// Mitsubishi GX Works2 project: CydeusPlatform   PLC: FX3U/FX3UC
// Cydeus Mitsu Platform

// global labels: GVL_Main
VAR_GLOBAL
  bAlarmTrigger AT M0 : BOOL;
  bManualMode AT M1 : BOOL;
  bAutoMode AT M2 : BOOL;
  bStepMode AT M3 : BOOL;
END_VAR

// global labels: GVL_Alarm
VAR_GLOBAL
  bMachineError AT M400 : BOOL;
  arrError AT M410 : ARRAY [0..9] OF BOOL;
  bResetError AT M401 : BOOL;
END_VAR
VAR_GLOBAL CONSTANT
  uiNumErrMinus1 : INT := 9;
END_VAR

// global labels: GVL_Output
VAR_GLOBAL
  bPunchingOutput AT Y006 : BOOL;
  bPowerMotor AT Y007 : BOOL;
END_VAR

// global labels: GVL_HMI
VAR_GLOBAL
  btnPunchingOutput : BOOL;
  btnPowerMotor : BOOL;
  btnManualMode : BOOL;
  btnInitialize : BOOL;
  btnAutoMode : BOOL;
  btnAbort : BOOL;
  btnStepMode : BOOL;
  btnBack : BOOL;
  btnTest : BOOL;
  btnTestManualOn : BOOL;
  btnSetup : BOOL;
END_VAR

// task Task_01 (event TRUE, interval 0, priority 31): MAIN

PROGRAM MAIN
VAR
  fbErrorController : FB_ErrorController;
  fbOutputController : FB_OutputController;
  fbStateMachine : FB_StateMachine;
END_VAR
	(*Auto Mode & Step Mode*)
	
	
	(*Manual Mode*)
	(*fbManualMode()*);
	
	(*State Machine*)
	fbStateMachine();
	
	(*Error Controller*)
	fbErrorController();
	
	(*Output Controller*)
	fbOutputController();
END_PROGRAM

FUNCTION_BLOCK FB_ErrorController
VAR
  ii : INT;
END_VAR
(*Error Controller*)

(*Reset Errors*)
IF bResetError THEN
	FOR ii := 0 TO uiNumErrMinus1  DO
		arrError[ii] := FALSE;
	END_FOR;
END_IF;

(*Register Errors*)
SET(bAlarmTrigger, arrError[0]);

(*Machine Error Trigger*)
bMachineError := FALSE;
FOR ii := 0 TO uiNumErrMinus1  DO
	bMachineError := bMachineError OR arrError[ii];
END_FOR;
END_FUNCTION_BLOCK

FUNCTION_BLOCK FB_OutputController
(*Output Controller*)

(*Calculate the logical output, then assign to physical output*)
bPowerMotor := FUN_Output();
bPunchingOutput := FUN_Output();
END_FUNCTION_BLOCK

FUNCTION_BLOCK FB_ManualMode
VAR_INPUT
  bEnable : BOOL;
END_VAR
(*Manual Mode*)

(*Enable Manual Mode*)
objPowerMotor.b_ManualMode := bManualMode;
objPunchingOutput.b_ManualMode := bManualMode;

(*Buttons on HMI control logical outputs*)
IF bManualMode THEN
	objPowerMotor.b_OutMan := btnPowerMotor;
	objPunchingOutput.b_OutMan := btnPunchingOutput;
END_IF;
END_FUNCTION_BLOCK

FUNCTION_BLOCK FB_StateMachine
VAR
  iState : INT;
  fbInitializing : FB_StateInitializing;
  fbAutoMode : FB_StateRunningAuto;
  fbManualMode : FB_ManualMode;
  iLastState : INT;
  bInitializingDone : BOOL;
  bAutoModeReturn : BOOL;
  bManualModeReturn : BOOL;
END_VAR
(*Main State Machine*)
IF (btnAbort OR bMachineError) AND NOT (iState = 1) AND NOT (iState >= 10) THEN	(*Abort command*)
	iState := 0;
END_IF;

CASE iState OF
	0: 		(*Aborting*)
		iState := 1;
	
	1: 		(*Begin*)
		IF btnInitialize AND NOT bMachineError THEN
			iState := 2;
		ELSIF btnTest THEN
			iLastState := iState;
			iState := 10;
		ELSIF btnSetup THEN
			iLastState := iState;
			iState := 15;
		END_IF;
		
	2: 		(*Initializing*)
		IF bInitializingDone AND NOT bMachineError THEN
			iState := 3;
		END_IF;
		
	3: 		(*Ready*)
		IF btnAutoMode AND NOT bMachineError THEN
			iState := 4;
		ELSIF btnStepMode AND NOT bMachineError THEN
			iState := 5;
		ELSIF btnManualMode AND NOT bMachineError THEN
			iState := 6;
		ELSIF btnTest THEN
			iLastState := iState;
			iState := 10;
		END_IF;
	
	4: 		(*Running Auto Mode*)
		IF bAutoModeReturn  AND NOT bMachineError THEN
			iState := 3;
		END_IF;
		
	5: 		(*Running Step Mode*)
		IF bAutoModeReturn AND NOT bMachineError THEN
			iState := 3;
		END_IF;
		
	6: 		(*Running Manual Mode*)
		IF btnBack AND NOT bMachineError THEN
			iState := 3;
		END_IF;
		
	10: 		(*Testing*)
		IF btnBack THEN
			iState := iLastState;
		END_IF;
		
	15: 		(*Setting*)
		IF btnBack THEN
			iState := iLastState;
		END_IF;
	
ELSE 
		;
END_CASE;

(*State Action*)
bAutoMode := iState = 4;
bStepMode := iState = 5;
bManualMode := iState = 6;

(*Function Block Call*)
fbInitializing(bEnable := iState = 2);
fbAutoMode(bEnable := (iState = 4) OR (iState = 5),
							bEnStepMode := iState = 5);
fbManualMode(bEnable := (iState = 6) OR (iState = 10 AND btnTestManualOn));

bAutoModeReturn := fbAutoMode.bReturn;
bInitializingDone := fbInitializing.bDone;
END_FUNCTION_BLOCK

FUNCTION_BLOCK FB_StateInitializing
VAR_OUTPUT
  bDone : BOOL;
END_VAR
VAR_INPUT
  bEnable : BOOL;
END_VAR
;
END_FUNCTION_BLOCK

FUNCTION_BLOCK FB_StateRunningAuto
VAR_OUTPUT
  bReturn : BOOL;
END_VAR
VAR_INPUT
  bEnStepMode : BOOL;
  bEnable : BOOL;
END_VAR
;
END_FUNCTION_BLOCK

FUNCTION FUN_Output
VAR_INPUT
  b_OutAuto : BOOL;
  b_OutMan : BOOL;
  b_ManualMode : BOOL;
END_VAR
FUN_Output := (b_ManualMode AND b_OutMan) OR (NOT b_ManualMode AND b_OutAuto);
END_FUNCTION

FUNCTION_BLOCK CL_1Sol2SenCylinder
VAR_INPUT
  biSensorActive : BOOL;
  biSensorHome : BOOL;
  bGoActive : BOOL;
  bReset : BOOL;
END_VAR
VAR_OUTPUT
  boSolenoid : BOOL;
  bBusy : BOOL;
  bInHomePos : BOOL;
  bInActivePos : BOOL;
  bError : BOOL;
END_VAR
VAR_INPUT
  tDelayTime : TIME;
  tTimeout : TIME;
END_VAR
VAR
  fbDelayTime : TON;
  fbTimeout : TON;
END_VAR
VAR_INPUT
  biActiveFeedback : BOOL;
END_VAR
(*Activate Output: Enable solenoid on valve*) 
boSolenoid := bGoActive;

(*Process Input: Wait for sensors signal*)
bInHomePos := fbDelayTime.Q AND biSensorHome AND NOT biSensorActive;
bInActivePos := fbDelayTime.Q AND biSensorActive AND NOT biSensorHome;
bBusy := (biActiveFeedback AND (biSensorHome OR NOT biSensorActive)) 
					OR (NOT biActiveFeedback AND (NOT biSensorHome OR biSensorActive));

(*Error handling*)
		(*Notify timeout error*)
		SET(fbTimeout.Q, bError);
		
		(*Reset timeout error*)
		RST(bReset, bError);

(*Timers call*)
fbDelayTime(IN := NOT bBusy, PT := tDelayTime);
fbTimeout(IN := bBusy, PT := tTimeout);
END_FUNCTION_BLOCK

FUNCTION_BLOCK CL_ServoMotor2
VAR_INPUT
  biINP : BOOL;
  biRD : BOOL;
  biALM : BOOL;
  bEnable : BOOL;
  bStop : BOOL;
  bAbort : BOOL;
  bReset : BOOL;
  bJogPos : BOOL;
  bJogNeg : BOOL;
  rJogDist : REAL;
  bMoveRel : BOOL;
  rMoveDist : REAL;
END_VAR
VAR_OUTPUT
  boNPz : BOOL;
  boCR : BOOL;
  boEM2 : BOOL;
  boSON : BOOL;
  boRES : BOOL;
  bBusy : BOOL;
  bError : BOOL;
  bDone : BOOL;
  bServoEnabled : BOOL;
END_VAR
VAR
  iState : INT;
  fbResetHold : TP_10;
  bResetHold : BOOL;
  fbMoveDelay : TON;
END_VAR
VAR_INPUT
  iMoveDelay : WORD;
END_VAR
VAR
  tMoveDelay : TIME;
  iStopState : INT;
END_VAR
VAR_INPUT
  iMoveVel : DINT;
  iMoveAccel : DINT;
  iPulsePerRev : DINT;
END_VAR
VAR
  rRadius : REAL;
  iFrequency : DINT;
  iPulse : DINT;
  iAccel : DINT;
  bOutPulse : BOOL;
END_VAR
VAR_INPUT
  iOutChannel : INT;
END_VAR
(*Procedure*)
		(*Abort*)
		IF bAbort OR NOT bEnable THEN
				iState := 0;
				iStopState := 0;
		END_IF;
		
		(*Reset*)
		IF bReset AND bError THEN
				iState := 0;
				iStopState := 0;
		END_IF;		
		
		(*Stop*)
		CASE iStopState OF
				0: 	(*Wait for stop signal*)
						IF bStop THEN
								iStopState := 10;
						END_IF;
						
				10: 	(*Execute Stop*)
						IF iState > 20 THEN
								iState := 20;
						END_IF;
						IF biINP THEN
								iStopState := 20;
						END_IF;
						
				20: 	(*Stop done, wait for command release*)
						IF NOT bStop THEN
								iStopState := 0;
						END_IF;
		END_CASE;	
						

(*Main State Machine*)
CASE iState OF 
		0: 	(*Unenabled, wait for Enable command*)
				IF bEnable AND NOT bStop AND NOT bError THEN
						iState := 10;
				END_IF;
				
		10: 	(*Servo On*)
				IF bServoEnabled THEN
						iState := 20;
				END_IF;
						
		20: 	(*Servo Ready, wait for moving command*)
				IF bJogPos AND NOT bStop AND NOT bError THEN
						iState := 100;
				ELSIF bJogNeg AND NOT bStop AND NOT bError THEN
						iState := 150;
				ELSIF bMoveRel AND NOT bStop AND NOT bError THEN
						iState := 200;
				END_IF;
				
		100: 	(*Calculate number of pulse*)			
				iFrequency := iPulsePerRev;
				iPulse := 0;	
				iState := 110;
				
		110: 	(*Execute Jog Pos command*)
				IF NOT bJogPos THEN 
						iState := 20;
				END_IF;
				
		150: 	(*Execute Jog Neg command*)
				IF NOT bJogNeg THEN
						iState := 20;
				END_IF;
				
		200: 	(*Calculate number of pulse*)
				iFrequency := REAL_TO_DINT(DINT_TO_REAL(iPulsePerRev*iMoveVel)/60.0);
				iPulse := REAL_TO_DINT(DINT_TO_REAL(iPulsePerRev)*rMoveDist/(2.0*3.1415926*rRadius));	
				iAccel := iMoveAccel;
				tMoveDelay := WORD_TO_TIME(iMoveDelay);
				iState := 210;
		
		210: 	(*Execute Move Relative command*)
				IF biINP AND fbMoveDelay.Q THEN
						iState := 220;
				END_IF;		
				
		220: 	(*Move Relative done, wait for command release*)
				IF NOT bMoveRel THEN
						iState := 20;
				END_IF;
				
END_CASE;
	
(*State Action*)
		boSON := (bEnable AND iState >= 10 AND NOT bAbort);			(*Enable Servo Motor*)	
		boEM2 := NOT bAbort;																			(*Abort Servo Motor*)
		boRES := fbResetHold.Q AND NOT biALM;									(*Reset Servo Motor*)		
		
		bBusy := (iState = 100) OR (iState = 150) OR (iState = 210) OR (iStopState = 10);
		bDone := (iState = 220) OR (iStopState = 20);									(*Servo movement is done*)
		bServoEnabled := biRD;																		(*Servo is powered on*)
	
		SET(NOT biALM, bError);																		(*Notify Servo Motor Error*)
		RST((bReset AND bError), bError);													(*Reset object error*)	
		
		bOutPulse := ((iState = 100) OR (iState = 150) OR (iState = 210)) AND NOT (iStopState = 10);	(*Enable Pulse*)
		boNPz := ((iState = 150) OR (rMoveDist < 0.0));
	
(*Function Block Call*)
PLS(bReset, bResetHold);
fbResetHold(IN := bResetHold, PT := t#60ms);
fbMoveDelay(IN := bMoveRel, PT := tMoveDelay);

CASE iOutChannel OF 
		0: 	(*Y000*)
				DPLSR(bOutPulse, iFrequency, iPulse, iAccel, Y000);
		1:		(*Y001*)
				DPLSR(bOutPulse, iFrequency, iPulse, iAccel, Y001);
		2:		(*Y002*)
				DPLSR(bOutPulse, iFrequency, iPulse, iAccel, Y002);
END_CASE;
END_FUNCTION_BLOCK

FUNCTION_BLOCK CL_ServoMotor
VAR_INPUT
  biINP : BOOL;
  biRD : BOOL;
  biALM : BOOL;
  bEnable : BOOL;
  bStop : BOOL;
  bAbort : BOOL;
  bReset : BOOL;
  bJogPos : BOOL;
  bJogNeg : BOOL;
  rJogDist : REAL;
  bMoveRel : BOOL;
  rMoveDist : REAL;
END_VAR
VAR_OUTPUT
  boNPz : BOOL;
  boCR : BOOL;
  boEM2 : BOOL;
  boSON : BOOL;
  boRES : BOOL;
  bBusy : BOOL;
  bError : BOOL;
  bDone : BOOL;
  bServoEnabled : BOOL;
END_VAR
VAR
  iState : INT;
  fbResetHold : TP_10;
  bResetHold : BOOL;
  fbMoveDelay : TON;
END_VAR
VAR_INPUT
  iMoveDelay : WORD;
END_VAR
VAR
  tMoveDelay : TIME;
  iStopState : INT;
END_VAR
VAR_INPUT
  iMoveVel : DINT;
  iMoveAccel : DINT;
  iPulsePerRev : DINT;
END_VAR
VAR
  rRadius : REAL;
  iFrequency : DINT;
  iPulse : DINT;
  iAccel : DINT;
  bOutPulse : BOOL;
END_VAR
VAR_INPUT
  iOutChannel : INT;
END_VAR
VAR
  bInJogPos : BOOL;
  bInJogNeg : BOOL;
  bInMoveRel : BOOL;
  iTestJog : INT;
  iTestMove : INT;
  bInEnabled : BOOL;
END_VAR
(*Procedure*)
		(*Abort*)
		IF bAbort OR NOT bEnable THEN
				iState := 0;
				iStopState := 0;
		END_IF;
		
		(*Reset*)
		IF bReset AND bError THEN
				iState := 0;
				iStopState := 0;
		END_IF;		
		
		(*Stop*)
		CASE iStopState OF
				0: 	(*Wait for stop signal*)
						IF bStop THEN
								iStopState := 10;
						END_IF;
						
				10: 	(*Execute Stop*)
						IF iState > 20 THEN
								iState := 20;
						END_IF;
						IF biINP THEN
								iStopState := 20;
						END_IF;
						
				20: 	(*Stop done, wait for command release*)
						IF NOT bStop THEN
								iStopState := 0;
						END_IF;
		END_CASE;	
						

(*Main State Machine*)
CASE iState OF 
		0: 	(*Unenabled, wait for Enable command*)
				IF bEnable AND NOT bStop AND NOT bError THEN
						iState := 10;
				END_IF;
				
		10: 	(*Servo On*)
				IF bServoEnabled THEN
						iState := 20;
				END_IF;
						
		20: 	(*Servo Ready, wait for moving command*)
				IF bJogPos AND NOT bStop AND NOT bError THEN
						iState := 100;
				ELSIF bJogNeg AND NOT bStop AND NOT bError THEN
						iState := 150;
				ELSIF bMoveRel AND NOT bStop AND NOT bError THEN
						iState := 200;
				END_IF;
				
		100: 	(*Calculate number of pulse*)			
				iFrequency := iPulsePerRev;
				iPulse := 0;	
				iState := 110;
				
		110: 	(*Execute Jog Pos command*)
				IF NOT bJogPos THEN 
						iState := 20;
				END_IF;
				
		150: 	(*Execute Jog Neg command*)
				IF NOT bJogNeg THEN
						iState := 20;
				END_IF;
				
		200: 	(*Calculate number of pulse*)
				iFrequency := REAL_TO_DINT(DINT_TO_REAL(iPulsePerRev*iMoveVel)/60.0);
				iPulse := REAL_TO_DINT(DINT_TO_REAL(iPulsePerRev)*rMoveDist/(2.0*3.1415926*rRadius));	
				iAccel := iMoveAccel;
				tMoveDelay := WORD_TO_TIME(iMoveDelay);
				iState := 210;
		
		210: 	(*Execute Move Relative command*)
				IF biINP AND fbMoveDelay.Q THEN
						iState := 220;
				END_IF;		
				
		220: 	(*Move Relative done, wait for command release*)
				IF NOT bMoveRel THEN
						iState := 20;
				END_IF;
				
END_CASE;
	

(*Activate Output*)
		(*Physical Output*)
		boSON := bInEnabled																				(*Enable Servo Motor*)	
		boEM2 := NOT bAbort;																			(*Abort Servo Motor*)
		boRES := fbResetHold.Q AND NOT biALM;									(*Reset Servo Motor*)		
		
		bBusy := bInJogPos OR bInJogNeg OR (bInMoveRel AND NOT (biINP AND fbMoveDelay.Q)) OR (bStop AND NOT biINP);
		bDone := (iState = 220) OR (iStopState = 20);									(*Servo movement is done*)
		bServoEnabled := biRD;																		(*Servo is powered on*)
	
		SET(NOT biALM, bError);																		(*Notify Servo Motor Error*)
		RST((bReset AND bError), bError);													(*Reset object error*)	
		
		bOutPulse := bInJogPos OR bInJogNeg OR (bInMoveRel AND NOT (biINP AND fbMoveDelay.Q));
		boNPz := ((iState = 150) OR (rMoveDist < 0.0));
		
(*Execute Moving function*)
		(*Enable*)
		bInEnabled := (bEnable AND NOT bAbort);	

		(*Jog command*)
		IF (bJogPos OR bJogNeg) AND NOT bBusy THEN
				iFrequency := iPulsePerRev;
				iPulse := 0;	
				iAccel := iMoveAccel;
				iTestJog := iTestJog + 1;
		END_IF;
		
		bInJogPos := bJogPos AND NOT bInJogNeg AND NOT bInMoveRel AND NOT bStop AND NOT bAbort;
		bInJogNeg := bJogNeg AND NOT bInJogPos AND NOT bInMoveRel AND NOT bStop AND NOT bAbort;
		
		(*Move Relative command*)
		IF bMoveRel AND NOT bBusy THEN
				iFrequency := REAL_TO_DINT(DINT_TO_REAL(iPulsePerRev*iMoveVel)/60.0);
				iPulse := REAL_TO_DINT(DINT_TO_REAL(iPulsePerRev)*rMoveDist/(2.0*3.1415926*rRadius));	
				iAccel := iMoveAccel;
				tMoveDelay := WORD_TO_TIME(iMoveDelay);
				iTestMove := iTestMove + 1;
		END_IF;
		
		bInMoveRel := bMoveRel AND NOT bInJogPos AND NOT bInJogNeg AND NOT bStop AND NOT bAbort;

		(*Output PTO*)
		CASE iOutChannel OF 
				0: 	(*Y000*)
						DPLSR(bOutPulse, iFrequency, iPulse, iAccel, Y000);
				1:		(*Y001*)
						DPLSR(bOutPulse, iFrequency, iPulse, iAccel, Y001);
				2:		(*Y002*)
						DPLSR(bOutPulse, iFrequency, iPulse, iAccel, Y002);
		END_CASE;
		
(*Function Block Call*)
PLS(bReset, bResetHold);
fbResetHold(IN := bResetHold, PT := t#60ms);
fbMoveDelay(IN := bMoveRel, PT := tMoveDelay);
END_FUNCTION_BLOCK
